// LS Electric XG5000 project: 동남133
// PLC NewPLC
// module base 0 slot 0: 입출력 모듈:XBC-DN/DP14E (DC 24V 입력 8점, 트랜지스터 출력 6점)

PROGRAM NewProgram (task: 스캔 프로그램)

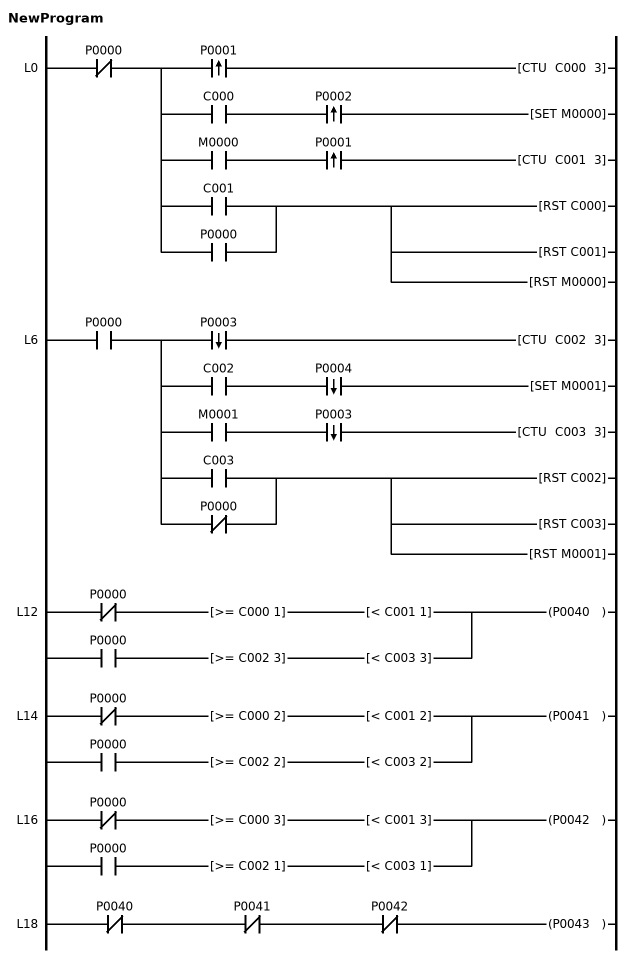
; L0
LOAD NOT  P0000
MPUSH
ANDP      P0001
CTU       C000 3
MLOAD
AND       C000
ANDP      P0002
SET       M0000
MLOAD
AND       M0000
ANDP      P0001
CTU       C001 3
MPOP
LOAD      C001
OR        P0000
AND LOAD
RST       C000
RST       C001
RST       M0000
; L6
LOAD      P0000
MPUSH
ANDN      P0003
CTU       C002 3
MLOAD
AND       C002
ANDN      P0004
SET       M0001
MLOAD
AND       M0001
ANDN      P0003
CTU       C003 3
MPOP
LOAD      C003
OR NOT    P0000
AND LOAD
RST       C002
RST       C003
RST       M0001
; L12
LOAD NOT  P0000
AND>=     C000 1
AND<      C001 1
LOAD      P0000
AND>=     C002 3
AND<      C003 3
OR LOAD
OUT       P0040
; L14
LOAD NOT  P0000
AND>=     C000 2
AND<      C001 2
LOAD      P0000
AND>=     C002 2
AND<      C003 2
OR LOAD
OUT       P0041
; L16
LOAD NOT  P0000
AND>=     C000 3
AND<      C001 3
LOAD      P0000
AND>=     C002 1
AND<      C003 1
OR LOAD
OUT       P0042
; L18
LOAD NOT  P0040
AND NOT   P0041
AND NOT   P0042
OUT       P0043